TYPE ST_HMI_Monitor_PSB :
STRUCT
	b_Connected : BOOL;
	b_Active	: BOOL;
END_STRUCT
END_TYPE

(* stored: Version 1.1.0.1, ProductVersion 3.1.4026.18
   DUT ST_HMI_Monitor_PSB: Id {dd5994a8-98f1-4d0b-b4c4-4e209700f1ff} *)
